{attribute 'qualified_only'}
{attribute 'strict'}
{attribute 'to_string'}
TYPE
ST140_Measure_e :
(
    RESET := 0, // Reset

    INIT := 100, // Initialisieren 

    READY := 999,  // READY to Start, Init Done 
    START := 1000, // Start Zyklisch

    waitOnMover,     // wait until the mover is there
    MOVER_NEEDED_OP, // Ab here, a mover in position is needed to perform the action

    Measure_right,
    Move_shuttle_relative_right,
    Move_shuttle_to_pos_left,
    Measure_left,
    Move_shuttle_relative_left,
    Save_result_in_mover,

    SYNC_MOVER_LEAVE, // MoverMan need to take the mover
    MOVER_FREE_OP,    // here, operation without mover can be done.

    DONE := 8000,  // Ablauf beendet 
    ERROR := 9000, // Fehler 
    _max
);
END_TYPE

(*
back to shuttle
check level NIO Box
*)

(* stored: Version 1.1.0.1, ProductVersion 3.1.4024.6
   EnumerationTextList ST140_Measure_e: Id {3f1e7fd2-5bdd-480c-b5e4-6a2be9165882} *)
